Fanuc KAREL source: DAQ_WRITE.kl

PROGRAM T
%NOLOCKGROUP
VAR
 v0 : INTEGER
 v1 : STRING[40]
 v2 : STRING[40]
 v3 : INTEGER
BEGIN
 DAQ_WRITE(v0, v1, v2, v3)
END T
